// C = A - B;
FUNCTION matSub : BOOL
VAR_IN_OUT CONSTANT
	matA :ARRAY[*,*] OF LREAL;
	matB :ARRAY[*,*] OF LREAL;
END_VAR

VAR_IN_OUT 
	matC :ARRAY[*,*] OF LREAL;
END_VAR

VAR
	m,n :DINT;
	i,j, k :DINT;
 
END_VAR

m:=UPPER_BOUND(matC,1);
n:= UPPER_BOUND(matC,2);
FOR i:=1 TO m DO
	FOR j:=1 TO n DO
		matC[i,j]:=matA[i,j]-matB[i,j];
	END_FOR
END_FOR

END_FUNCTION

(* stored: Version 1.1.0.1, ProductVersion 3.1.4024.12
   POU matSub: Id {39727f23-bf8c-437d-94a5-9f9adefa65d5}, SpecialFunc None *)
